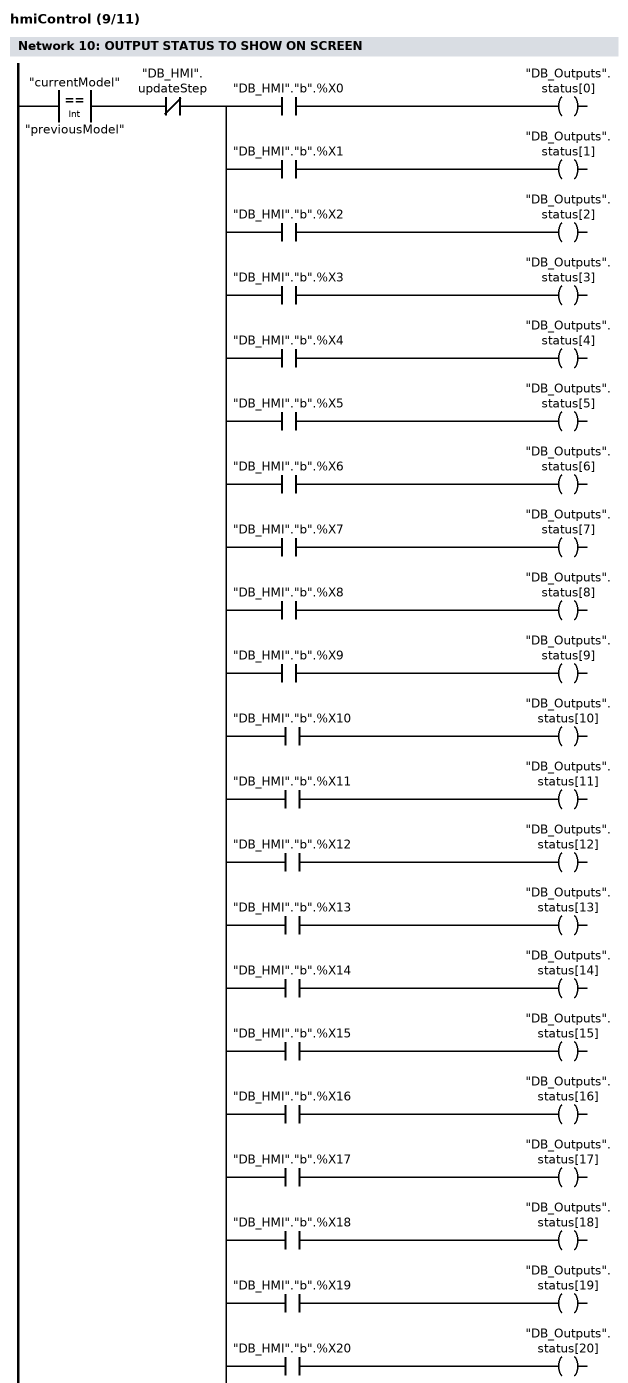
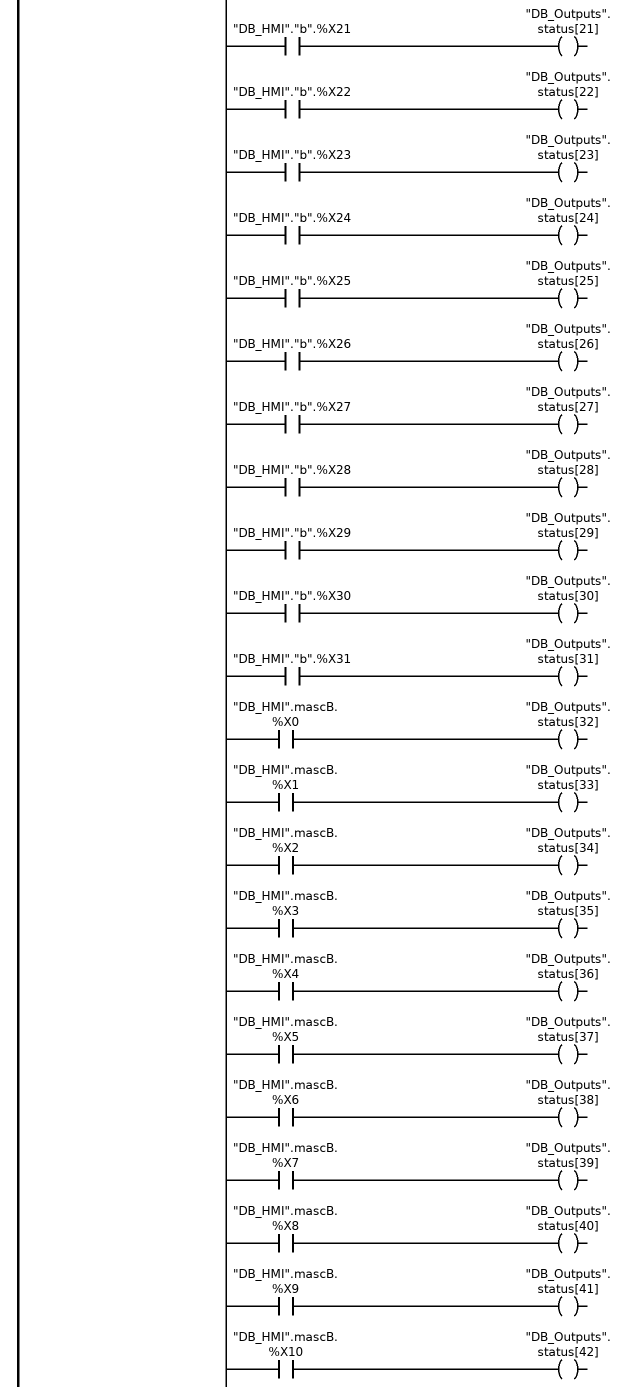
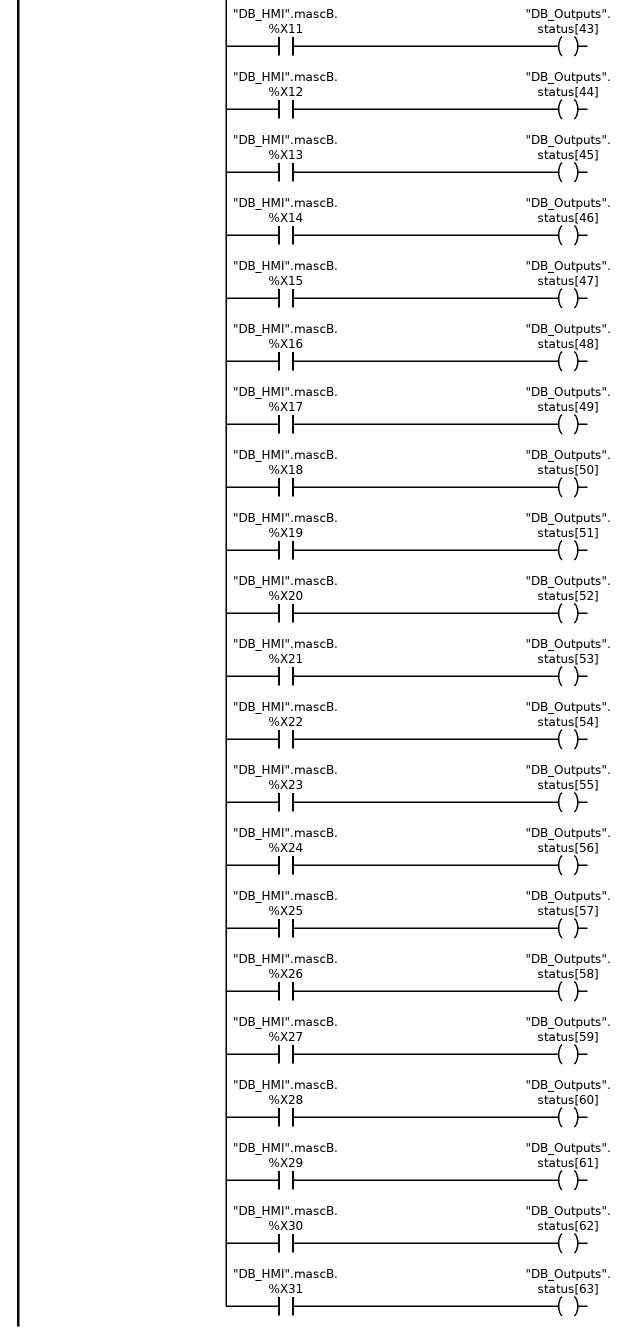
   RUNG wire#powerrail
      { S7_Templates := "SrcType := Int" } EQ_Contact(in1 := "currentModel", in2 := "previousModel")
      I_Contact( "DB_HMI".updateStep )
      wire#w1
      Contact( "DB_HMI"."b".%X0 )
      Coil( "DB_Outputs".status[0] )
   END_RUNG
   RUNG wire#w1
      Contact( "DB_HMI"."b".%X1 )
      Coil( "DB_Outputs".status[1] )
   END_RUNG
   RUNG wire#w1
      Contact( "DB_HMI"."b".%X2 )
      Coil( "DB_Outputs".status[2] )
   END_RUNG
   RUNG wire#w1
      Contact( "DB_HMI"."b".%X3 )
      Coil( "DB_Outputs".status[3] )
   END_RUNG
   RUNG wire#w1
      Contact( "DB_HMI"."b".%X4 )
      Coil( "DB_Outputs".status[4] )
   END_RUNG
   RUNG wire#w1
      Contact( "DB_HMI"."b".%X5 )
      Coil( "DB_Outputs".status[5] )
   END_RUNG
   RUNG wire#w1
      Contact( "DB_HMI"."b".%X6 )
      Coil( "DB_Outputs".status[6] )
   END_RUNG
   RUNG wire#w1
      Contact( "DB_HMI"."b".%X7 )
      Coil( "DB_Outputs".status[7] )
   END_RUNG
   RUNG wire#w1
      Contact( "DB_HMI"."b".%X8 )
      Coil( "DB_Outputs".status[8] )
   END_RUNG
   RUNG wire#w1
      Contact( "DB_HMI"."b".%X9 )
      Coil( "DB_Outputs".status[9] )
   END_RUNG
   RUNG wire#w1
      Contact( "DB_HMI"."b".%X10 )
      Coil( "DB_Outputs".status[10] )
   END_RUNG
   RUNG wire#w1
      Contact( "DB_HMI"."b".%X11 )
      Coil( "DB_Outputs".status[11] )
   END_RUNG
   RUNG wire#w1
      Contact( "DB_HMI"."b".%X12 )
      Coil( "DB_Outputs".status[12] )
   END_RUNG
   RUNG wire#w1
      Contact( "DB_HMI"."b".%X13 )
      Coil( "DB_Outputs".status[13] )
   END_RUNG
   RUNG wire#w1
      Contact( "DB_HMI"."b".%X14 )
      Coil( "DB_Outputs".status[14] )
   END_RUNG
   RUNG wire#w1
      Contact( "DB_HMI"."b".%X15 )
      Coil( "DB_Outputs".status[15] )
   END_RUNG
   RUNG wire#w1
      Contact( "DB_HMI"."b".%X16 )
      Coil( "DB_Outputs".status[16] )
   END_RUNG
   RUNG wire#w1
      Contact( "DB_HMI"."b".%X17 )
      Coil( "DB_Outputs".status[17] )
   END_RUNG
   RUNG wire#w1
      Contact( "DB_HMI"."b".%X18 )
      Coil( "DB_Outputs".status[18] )
   END_RUNG
   RUNG wire#w1
      Contact( "DB_HMI"."b".%X19 )
      Coil( "DB_Outputs".status[19] )
   END_RUNG
   RUNG wire#w1
      Contact( "DB_HMI"."b".%X20 )
      Coil( "DB_Outputs".status[20] )
   END_RUNG
   RUNG wire#w1
      Contact( "DB_HMI"."b".%X21 )
      Coil( "DB_Outputs".status[21] )
   END_RUNG
   RUNG wire#w1
      Contact( "DB_HMI"."b".%X22 )
      Coil( "DB_Outputs".status[22] )
   END_RUNG
   RUNG wire#w1
      Contact( "DB_HMI"."b".%X23 )
      Coil( "DB_Outputs".status[23] )
   END_RUNG
   RUNG wire#w1
      Contact( "DB_HMI"."b".%X24 )
      Coil( "DB_Outputs".status[24] )
   END_RUNG
   RUNG wire#w1
      Contact( "DB_HMI"."b".%X25 )
      Coil( "DB_Outputs".status[25] )
   END_RUNG
   RUNG wire#w1
      Contact( "DB_HMI"."b".%X26 )
      Coil( "DB_Outputs".status[26] )
   END_RUNG
   RUNG wire#w1
      Contact( "DB_HMI"."b".%X27 )
      Coil( "DB_Outputs".status[27] )
   END_RUNG
   RUNG wire#w1
      Contact( "DB_HMI"."b".%X28 )
      Coil( "DB_Outputs".status[28] )
   END_RUNG
   RUNG wire#w1
      Contact( "DB_HMI"."b".%X29 )
      Coil( "DB_Outputs".status[29] )
   END_RUNG
   RUNG wire#w1
      Contact( "DB_HMI"."b".%X30 )
      Coil( "DB_Outputs".status[30] )
   END_RUNG
   RUNG wire#w1
      Contact( "DB_HMI"."b".%X31 )
      Coil( "DB_Outputs".status[31] )
   END_RUNG
   RUNG wire#w1
      Contact( "DB_HMI".mascB.%X0 )
      Coil( "DB_Outputs".status[32] )
   END_RUNG
   RUNG wire#w1
      Contact( "DB_HMI".mascB.%X1 )
      Coil( "DB_Outputs".status[33] )
   END_RUNG
   RUNG wire#w1
      Contact( "DB_HMI".mascB.%X2 )
      Coil( "DB_Outputs".status[34] )
   END_RUNG
   RUNG wire#w1
      Contact( "DB_HMI".mascB.%X3 )
      Coil( "DB_Outputs".status[35] )
   END_RUNG
   RUNG wire#w1
      Contact( "DB_HMI".mascB.%X4 )
      Coil( "DB_Outputs".status[36] )
   END_RUNG
   RUNG wire#w1
      Contact( "DB_HMI".mascB.%X5 )
      Coil( "DB_Outputs".status[37] )
   END_RUNG
   RUNG wire#w1
      Contact( "DB_HMI".mascB.%X6 )
      Coil( "DB_Outputs".status[38] )
   END_RUNG
   RUNG wire#w1
      Contact( "DB_HMI".mascB.%X7 )
      Coil( "DB_Outputs".status[39] )
   END_RUNG
   RUNG wire#w1
      Contact( "DB_HMI".mascB.%X8 )
      Coil( "DB_Outputs".status[40] )
   END_RUNG
   RUNG wire#w1
      Contact( "DB_HMI".mascB.%X9 )
      Coil( "DB_Outputs".status[41] )
   END_RUNG
   RUNG wire#w1
      Contact( "DB_HMI".mascB.%X10 )
      Coil( "DB_Outputs".status[42] )
   END_RUNG
   RUNG wire#w1
      Contact( "DB_HMI".mascB.%X11 )
      Coil( "DB_Outputs".status[43] )
   END_RUNG
   RUNG wire#w1
      Contact( "DB_HMI".mascB.%X12 )
      Coil( "DB_Outputs".status[44] )
   END_RUNG
   RUNG wire#w1
      Contact( "DB_HMI".mascB.%X13 )
      Coil( "DB_Outputs".status[45] )
   END_RUNG
   RUNG wire#w1
      Contact( "DB_HMI".mascB.%X14 )
      Coil( "DB_Outputs".status[46] )
   END_RUNG
   RUNG wire#w1
      Contact( "DB_HMI".mascB.%X15 )
      Coil( "DB_Outputs".status[47] )
   END_RUNG
   RUNG wire#w1
      Contact( "DB_HMI".mascB.%X16 )
      Coil( "DB_Outputs".status[48] )
   END_RUNG
   RUNG wire#w1
      Contact( "DB_HMI".mascB.%X17 )
      Coil( "DB_Outputs".status[49] )
   END_RUNG
   RUNG wire#w1
      Contact( "DB_HMI".mascB.%X18 )
      Coil( "DB_Outputs".status[50] )
   END_RUNG
   RUNG wire#w1
      Contact( "DB_HMI".mascB.%X19 )
      Coil( "DB_Outputs".status[51] )
   END_RUNG
   RUNG wire#w1
      Contact( "DB_HMI".mascB.%X20 )
      Coil( "DB_Outputs".status[52] )
   END_RUNG
   RUNG wire#w1
      Contact( "DB_HMI".mascB.%X21 )
      Coil( "DB_Outputs".status[53] )
   END_RUNG
   RUNG wire#w1
      Contact( "DB_HMI".mascB.%X22 )
      Coil( "DB_Outputs".status[54] )
   END_RUNG
   RUNG wire#w1
      Contact( "DB_HMI".mascB.%X23 )
      Coil( "DB_Outputs".status[55] )
   END_RUNG
   RUNG wire#w1
      Contact( "DB_HMI".mascB.%X24 )
      Coil( "DB_Outputs".status[56] )
   END_RUNG
   RUNG wire#w1
      Contact( "DB_HMI".mascB.%X25 )
      Coil( "DB_Outputs".status[57] )
   END_RUNG
   RUNG wire#w1
      Contact( "DB_HMI".mascB.%X26 )
      Coil( "DB_Outputs".status[58] )
   END_RUNG
   RUNG wire#w1
      Contact( "DB_HMI".mascB.%X27 )
      Coil( "DB_Outputs".status[59] )
   END_RUNG
   RUNG wire#w1
      Contact( "DB_HMI".mascB.%X28 )
      Coil( "DB_Outputs".status[60] )
   END_RUNG
   RUNG wire#w1
      Contact( "DB_HMI".mascB.%X29 )
      Coil( "DB_Outputs".status[61] )
   END_RUNG
   RUNG wire#w1
      Contact( "DB_HMI".mascB.%X30 )
      Coil( "DB_Outputs".status[62] )
   END_RUNG
   RUNG wire#w1
      Contact( "DB_HMI".mascB.%X31 )
      Coil( "DB_Outputs".status[63] )
   END_RUNG
   // the same network as SCL:
   #_w1 := ("currentModel" = "previousModel") AND NOT "DB_HMI".updateStep;
   "DB_Outputs".status[0] := #_w1 AND "DB_HMI"."b".%X0;
   "DB_Outputs".status[1] := #_w1 AND "DB_HMI"."b".%X1;
   "DB_Outputs".status[2] := #_w1 AND "DB_HMI"."b".%X2;
   "DB_Outputs".status[3] := #_w1 AND "DB_HMI"."b".%X3;
   "DB_Outputs".status[4] := #_w1 AND "DB_HMI"."b".%X4;
   "DB_Outputs".status[5] := #_w1 AND "DB_HMI"."b".%X5;
   "DB_Outputs".status[6] := #_w1 AND "DB_HMI"."b".%X6;
   "DB_Outputs".status[7] := #_w1 AND "DB_HMI"."b".%X7;
   "DB_Outputs".status[8] := #_w1 AND "DB_HMI"."b".%X8;
   "DB_Outputs".status[9] := #_w1 AND "DB_HMI"."b".%X9;
   "DB_Outputs".status[10] := #_w1 AND "DB_HMI"."b".%X10;
   "DB_Outputs".status[11] := #_w1 AND "DB_HMI"."b".%X11;
   "DB_Outputs".status[12] := #_w1 AND "DB_HMI"."b".%X12;
   "DB_Outputs".status[13] := #_w1 AND "DB_HMI"."b".%X13;
   "DB_Outputs".status[14] := #_w1 AND "DB_HMI"."b".%X14;
   "DB_Outputs".status[15] := #_w1 AND "DB_HMI"."b".%X15;
   "DB_Outputs".status[16] := #_w1 AND "DB_HMI"."b".%X16;
   "DB_Outputs".status[17] := #_w1 AND "DB_HMI"."b".%X17;
   "DB_Outputs".status[18] := #_w1 AND "DB_HMI"."b".%X18;
   "DB_Outputs".status[19] := #_w1 AND "DB_HMI"."b".%X19;
   "DB_Outputs".status[20] := #_w1 AND "DB_HMI"."b".%X20;
   "DB_Outputs".status[21] := #_w1 AND "DB_HMI"."b".%X21;
   "DB_Outputs".status[22] := #_w1 AND "DB_HMI"."b".%X22;
   "DB_Outputs".status[23] := #_w1 AND "DB_HMI"."b".%X23;
   "DB_Outputs".status[24] := #_w1 AND "DB_HMI"."b".%X24;
   "DB_Outputs".status[25] := #_w1 AND "DB_HMI"."b".%X25;
   "DB_Outputs".status[26] := #_w1 AND "DB_HMI"."b".%X26;
   "DB_Outputs".status[27] := #_w1 AND "DB_HMI"."b".%X27;
   "DB_Outputs".status[28] := #_w1 AND "DB_HMI"."b".%X28;
   "DB_Outputs".status[29] := #_w1 AND "DB_HMI"."b".%X29;
   "DB_Outputs".status[30] := #_w1 AND "DB_HMI"."b".%X30;
   "DB_Outputs".status[31] := #_w1 AND "DB_HMI"."b".%X31;
   "DB_Outputs".status[32] := #_w1 AND "DB_HMI".mascB.%X0;
   "DB_Outputs".status[33] := #_w1 AND "DB_HMI".mascB.%X1;
   "DB_Outputs".status[34] := #_w1 AND "DB_HMI".mascB.%X2;
   "DB_Outputs".status[35] := #_w1 AND "DB_HMI".mascB.%X3;
   "DB_Outputs".status[36] := #_w1 AND "DB_HMI".mascB.%X4;
   "DB_Outputs".status[37] := #_w1 AND "DB_HMI".mascB.%X5;
   "DB_Outputs".status[38] := #_w1 AND "DB_HMI".mascB.%X6;
   "DB_Outputs".status[39] := #_w1 AND "DB_HMI".mascB.%X7;
   "DB_Outputs".status[40] := #_w1 AND "DB_HMI".mascB.%X8;
   "DB_Outputs".status[41] := #_w1 AND "DB_HMI".mascB.%X9;
   "DB_Outputs".status[42] := #_w1 AND "DB_HMI".mascB.%X10;
   "DB_Outputs".status[43] := #_w1 AND "DB_HMI".mascB.%X11;
   "DB_Outputs".status[44] := #_w1 AND "DB_HMI".mascB.%X12;
   "DB_Outputs".status[45] := #_w1 AND "DB_HMI".mascB.%X13;
   "DB_Outputs".status[46] := #_w1 AND "DB_HMI".mascB.%X14;
   "DB_Outputs".status[47] := #_w1 AND "DB_HMI".mascB.%X15;
   "DB_Outputs".status[48] := #_w1 AND "DB_HMI".mascB.%X16;
   "DB_Outputs".status[49] := #_w1 AND "DB_HMI".mascB.%X17;
   "DB_Outputs".status[50] := #_w1 AND "DB_HMI".mascB.%X18;
   "DB_Outputs".status[51] := #_w1 AND "DB_HMI".mascB.%X19;
   "DB_Outputs".status[52] := #_w1 AND "DB_HMI".mascB.%X20;
   "DB_Outputs".status[53] := #_w1 AND "DB_HMI".mascB.%X21;
   "DB_Outputs".status[54] := #_w1 AND "DB_HMI".mascB.%X22;
   "DB_Outputs".status[55] := #_w1 AND "DB_HMI".mascB.%X23;
   "DB_Outputs".status[56] := #_w1 AND "DB_HMI".mascB.%X24;
   "DB_Outputs".status[57] := #_w1 AND "DB_HMI".mascB.%X25;
   "DB_Outputs".status[58] := #_w1 AND "DB_HMI".mascB.%X26;
   "DB_Outputs".status[59] := #_w1 AND "DB_HMI".mascB.%X27;
   "DB_Outputs".status[60] := #_w1 AND "DB_HMI".mascB.%X28;
   "DB_Outputs".status[61] := #_w1 AND "DB_HMI".mascB.%X29;
   "DB_Outputs".status[62] := #_w1 AND "DB_HMI".mascB.%X30;
   "DB_Outputs".status[63] := #_w1 AND "DB_HMI".mascB.%X31;
END_REGION

REGION Network 11: HOME BUTTON
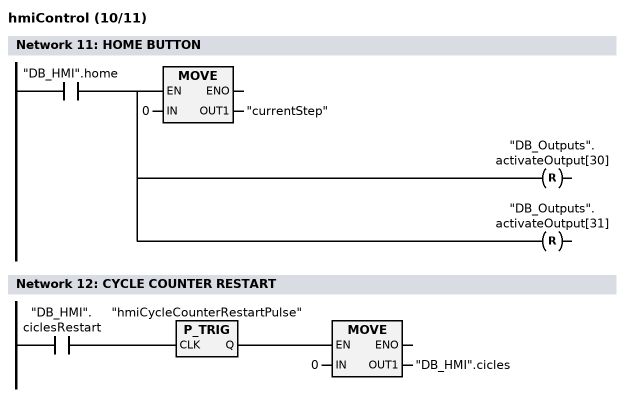
   RUNG wire#powerrail
      Contact( "DB_HMI".home )
      wire#w1
      Move(in := 0, out1 => "currentStep")
   END_RUNG
   RUNG wire#w1
      R_Coil( "DB_Outputs".activateOutput[30] )
   END_RUNG
   RUNG wire#w1
      R_Coil( "DB_Outputs".activateOutput[31] )
   END_RUNG
   // the same network as SCL:
   IF "DB_HMI".home THEN
       "currentStep" := 0;
       "DB_Outputs".activateOutput[30] := FALSE;
       "DB_Outputs".activateOutput[31] := FALSE;
   END_IF;
END_REGION

REGION Network 12: CYCLE COUNTER RESTART
   RUNG wire#powerrail
      Contact( "DB_HMI".ciclesRestart )
      P_Trig( "hmiCycleCounterRestartPulse" )
      Move(in := 0, out1 => "DB_HMI".cicles)
   END_RUNG
   // the same network as SCL:
   #_w1 := "DB_HMI".ciclesRestart AND NOT "hmiCycleCounterRestartPulse";   // rising edge
   "hmiCycleCounterRestartPulse" := "DB_HMI".ciclesRestart;
   IF #_w1 THEN "DB_HMI".cicles := 0; END_IF;
END_REGION

REGION Network 13: MODEL SELECTION
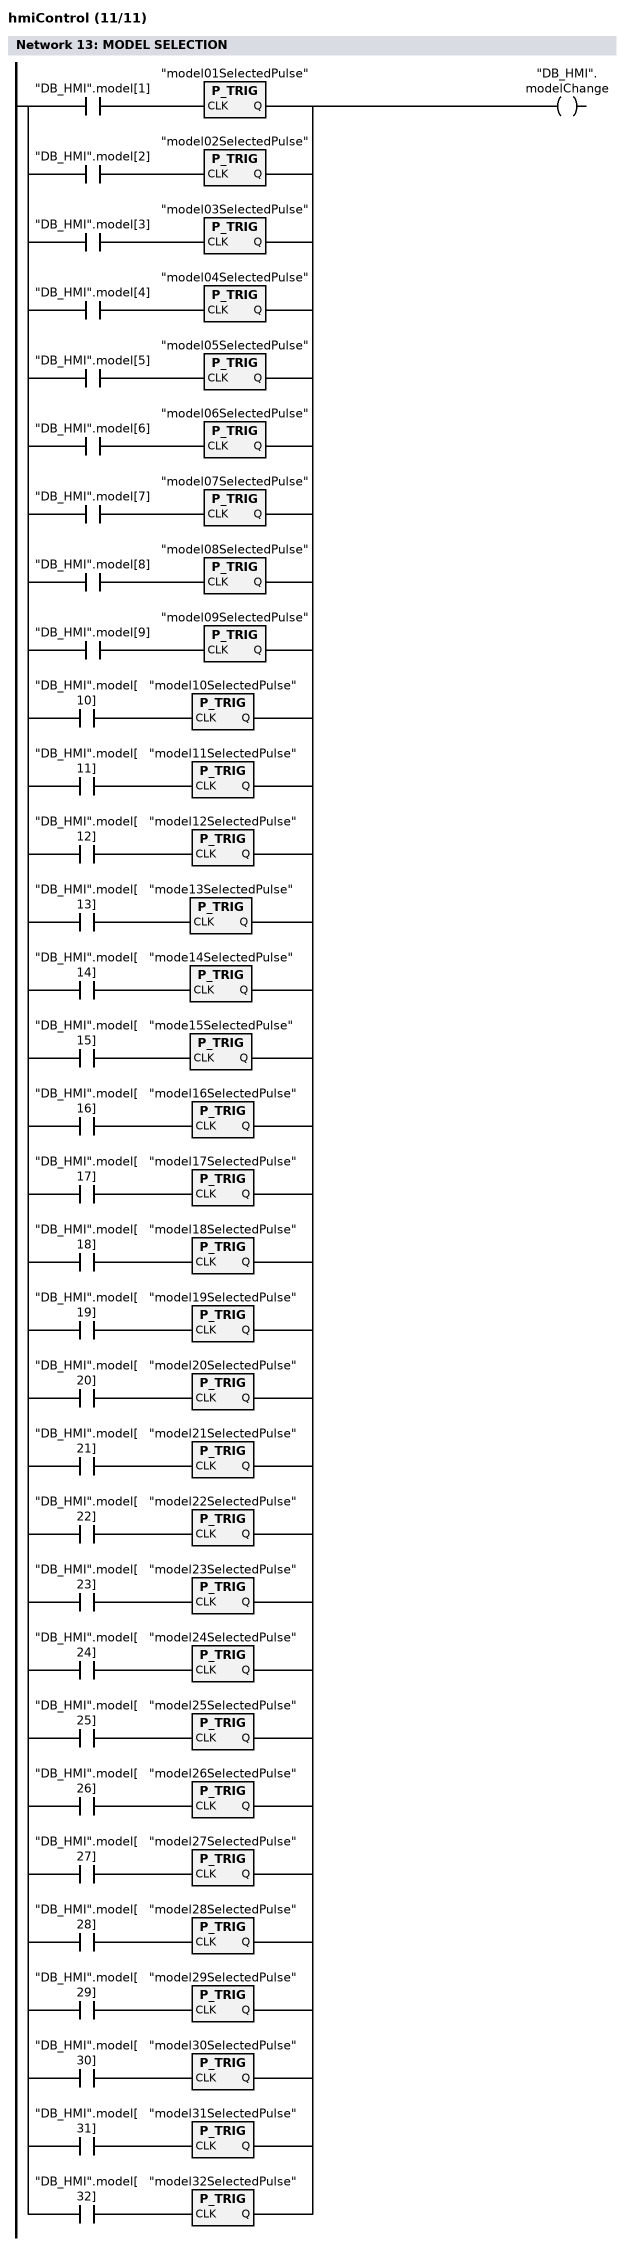
   RUNG wire#powerrail
      Contact( "DB_HMI".model[1] )
      P_Trig( "model01SelectedPulse" )
      wire#w1
      Coil( "DB_HMI".modelChange )
   END_RUNG
   RUNG wire#powerrail
      Contact( "DB_HMI".model[2] )
      P_Trig( "model02SelectedPulse" )
   END_RUNG wire#w1
   RUNG wire#powerrail
      Contact( "DB_HMI".model[3] )
      P_Trig( "model03SelectedPulse" )
   END_RUNG wire#w1
   RUNG wire#powerrail
      Contact( "DB_HMI".model[4] )
      P_Trig( "model04SelectedPulse" )
   END_RUNG wire#w1
   RUNG wire#powerrail
      Contact( "DB_HMI".model[5] )
      P_Trig( "model05SelectedPulse" )
   END_RUNG wire#w1
   RUNG wire#powerrail
      Contact( "DB_HMI".model[6] )
      P_Trig( "model06SelectedPulse" )
   END_RUNG wire#w1
   RUNG wire#powerrail
      Contact( "DB_HMI".model[7] )
      P_Trig( "model07SelectedPulse" )
   END_RUNG wire#w1
   RUNG wire#powerrail
      Contact( "DB_HMI".model[8] )
      P_Trig( "model08SelectedPulse" )
   END_RUNG wire#w1
   RUNG wire#powerrail
      Contact( "DB_HMI".model[9] )
      P_Trig( "model09SelectedPulse" )
   END_RUNG wire#w1
   RUNG wire#powerrail
      Contact( "DB_HMI".model[10] )
      P_Trig( "model10SelectedPulse" )
   END_RUNG wire#w1
   RUNG wire#powerrail
      Contact( "DB_HMI".model[11] )
      P_Trig( "model11SelectedPulse" )
   END_RUNG wire#w1
   RUNG wire#powerrail
      Contact( "DB_HMI".model[12] )
      P_Trig( "model12SelectedPulse" )
   END_RUNG wire#w1
   RUNG wire#powerrail
      Contact( "DB_HMI".model[13] )
      P_Trig( "mode13SelectedPulse" )
   END_RUNG wire#w1
   RUNG wire#powerrail
      Contact( "DB_HMI".model[14] )
      P_Trig( "mode14SelectedPulse" )
   END_RUNG wire#w1
   RUNG wire#powerrail
      Contact( "DB_HMI".model[15] )
      P_Trig( "mode15SelectedPulse" )
   END_RUNG wire#w1
   RUNG wire#powerrail
      Contact( "DB_HMI".model[16] )
      P_Trig( "model16SelectedPulse" )
   END_RUNG wire#w1
   RUNG wire#powerrail
      Contact( "DB_HMI".model[17] )
      P_Trig( "model17SelectedPulse" )
   END_RUNG wire#w1
   RUNG wire#powerrail
      Contact( "DB_HMI".model[18] )
      P_Trig( "model18SelectedPulse" )
   END_RUNG wire#w1
   RUNG wire#powerrail
      Contact( "DB_HMI".model[19] )
      P_Trig( "model19SelectedPulse" )
   END_RUNG wire#w1
   RUNG wire#powerrail
      Contact( "DB_HMI".model[20] )
      P_Trig( "model20SelectedPulse" )
   END_RUNG wire#w1
   RUNG wire#powerrail
      Contact( "DB_HMI".model[21] )
      P_Trig( "model21SelectedPulse" )
   END_RUNG wire#w1
   RUNG wire#powerrail
      Contact( "DB_HMI".model[22] )
      P_Trig( "model22SelectedPulse" )
   END_RUNG wire#w1
   RUNG wire#powerrail
      Contact( "DB_HMI".model[23] )
      P_Trig( "model23SelectedPulse" )
   END_RUNG wire#w1
   RUNG wire#powerrail
      Contact( "DB_HMI".model[24] )
      P_Trig( "model24SelectedPulse" )
   END_RUNG wire#w1
   RUNG wire#powerrail
      Contact( "DB_HMI".model[25] )
      P_Trig( "model25SelectedPulse" )
   END_RUNG wire#w1
   RUNG wire#powerrail
      Contact( "DB_HMI".model[26] )
      P_Trig( "model26SelectedPulse" )
   END_RUNG wire#w1
   RUNG wire#powerrail
      Contact( "DB_HMI".model[27] )
      P_Trig( "model27SelectedPulse" )
   END_RUNG wire#w1
   RUNG wire#powerrail
      Contact( "DB_HMI".model[28] )
      P_Trig( "model28SelectedPulse" )
   END_RUNG wire#w1
   RUNG wire#powerrail
      Contact( "DB_HMI".model[29] )
      P_Trig( "model29SelectedPulse" )
   END_RUNG wire#w1
   RUNG wire#powerrail
      Contact( "DB_HMI".model[30] )
      P_Trig( "model30SelectedPulse" )
   END_RUNG wire#w1
   RUNG wire#powerrail
      Contact( "DB_HMI".model[31] )
      P_Trig( "model31SelectedPulse" )
   END_RUNG wire#w1
   RUNG wire#powerrail
      Contact( "DB_HMI".model[32] )
      P_Trig( "model32SelectedPulse" )
   END_RUNG wire#w1
   // the same network as SCL:
   #_w1 := "DB_HMI".model[1] AND NOT "model01SelectedPulse";   // rising edge
   "model01SelectedPulse" := "DB_HMI".model[1];
   #_w2 := "DB_HMI".model[2] AND NOT "model02SelectedPulse";   // rising edge
   "model02SelectedPulse" := "DB_HMI".model[2];
   #_w3 := "DB_HMI".model[3] AND NOT "model03SelectedPulse";   // rising edge
   "model03SelectedPulse" := "DB_HMI".model[3];
   #_w4 := "DB_HMI".model[4] AND NOT "model04SelectedPulse";   // rising edge
   "model04SelectedPulse" := "DB_HMI".model[4];
   #_w5 := "DB_HMI".model[5] AND NOT "model05SelectedPulse";   // rising edge
   "model05SelectedPulse" := "DB_HMI".model[5];
   #_w6 := "DB_HMI".model[6] AND NOT "model06SelectedPulse";   // rising edge
   "model06SelectedPulse" := "DB_HMI".model[6];
   #_w7 := "DB_HMI".model[7] AND NOT "model07SelectedPulse";   // rising edge
   "model07SelectedPulse" := "DB_HMI".model[7];
   #_w8 := "DB_HMI".model[8] AND NOT "model08SelectedPulse";   // rising edge
   "model08SelectedPulse" := "DB_HMI".model[8];
   #_w9 := "DB_HMI".model[9] AND NOT "model09SelectedPulse";   // rising edge
   "model09SelectedPulse" := "DB_HMI".model[9];
   #_w10 := "DB_HMI".model[10] AND NOT "model10SelectedPulse";   // rising edge
   "model10SelectedPulse" := "DB_HMI".model[10];
   #_w11 := "DB_HMI".model[11] AND NOT "model11SelectedPulse";   // rising edge
   "model11SelectedPulse" := "DB_HMI".model[11];
   #_w12 := "DB_HMI".model[12] AND NOT "model12SelectedPulse";   // rising edge
   "model12SelectedPulse" := "DB_HMI".model[12];
   #_w13 := "DB_HMI".model[13] AND NOT "mode13SelectedPulse";   // rising edge
   "mode13SelectedPulse" := "DB_HMI".model[13];
   #_w14 := "DB_HMI".model[14] AND NOT "mode14SelectedPulse";   // rising edge
   "mode14SelectedPulse" := "DB_HMI".model[14];
   #_w15 := "DB_HMI".model[15] AND NOT "mode15SelectedPulse";   // rising edge
   "mode15SelectedPulse" := "DB_HMI".model[15];
   #_w16 := "DB_HMI".model[16] AND NOT "model16SelectedPulse";   // rising edge
   "model16SelectedPulse" := "DB_HMI".model[16];
   #_w17 := "DB_HMI".model[17] AND NOT "model17SelectedPulse";   // rising edge
   "model17SelectedPulse" := "DB_HMI".model[17];
   #_w18 := "DB_HMI".model[18] AND NOT "model18SelectedPulse";   // rising edge
   "model18SelectedPulse" := "DB_HMI".model[18];
   #_w19 := "DB_HMI".model[19] AND NOT "model19SelectedPulse";   // rising edge
   "model19SelectedPulse" := "DB_HMI".model[19];
   #_w20 := "DB_HMI".model[20] AND NOT "model20SelectedPulse";   // rising edge
   "model20SelectedPulse" := "DB_HMI".model[20];
   #_w21 := "DB_HMI".model[21] AND NOT "model21SelectedPulse";   // rising edge
   "model21SelectedPulse" := "DB_HMI".model[21];
   #_w22 := "DB_HMI".model[22] AND NOT "model22SelectedPulse";   // rising edge
   "model22SelectedPulse" := "DB_HMI".model[22];
   #_w23 := "DB_HMI".model[23] AND NOT "model23SelectedPulse";   // rising edge
   "model23SelectedPulse" := "DB_HMI".model[23];
   #_w24 := "DB_HMI".model[24] AND NOT "model24SelectedPulse";   // rising edge
   "model24SelectedPulse" := "DB_HMI".model[24];
   #_w25 := "DB_HMI".model[25] AND NOT "model25SelectedPulse";   // rising edge
   "model25SelectedPulse" := "DB_HMI".model[25];
   #_w26 := "DB_HMI".model[26] AND NOT "model26SelectedPulse";   // rising edge
   "model26SelectedPulse" := "DB_HMI".model[26];
   #_w27 := "DB_HMI".model[27] AND NOT "model27SelectedPulse";   // rising edge
   "model27SelectedPulse" := "DB_HMI".model[27];
   #_w28 := "DB_HMI".model[28] AND NOT "model28SelectedPulse";   // rising edge
   "model28SelectedPulse" := "DB_HMI".model[28];
   #_w29 := "DB_HMI".model[29] AND NOT "model29SelectedPulse";   // rising edge
   "model29SelectedPulse" := "DB_HMI".model[29];
   #_w30 := "DB_HMI".model[30] AND NOT "model30SelectedPulse";   // rising edge
   "model30SelectedPulse" := "DB_HMI".model[30];
   #_w31 := "DB_HMI".model[31] AND NOT "model31SelectedPulse";   // rising edge
   "model31SelectedPulse" := "DB_HMI".model[31];
   #_w32 := "DB_HMI".model[32] AND NOT "model32SelectedPulse";   // rising edge
   "model32SelectedPulse" := "DB_HMI".model[32];
   "DB_HMI".modelChange := #_w1 OR #_w2 OR #_w3 OR #_w4 OR #_w5 OR #_w6 OR #_w7 OR #_w8 OR #_w9 OR #_w10 OR #_w11 OR #_w12 OR #_w13 OR #_w14 OR #_w15 OR #_w16 OR #_w17 OR #_w18 OR #_w19 OR #_w20 OR #_w21 OR #_w22 OR #_w23 OR #_w24 OR #_w25 OR #_w26 OR #_w27 OR #_w28 OR #_w29 OR #_w30 OR #_w31 OR #_w32;
END_REGION
END_FUNCTION
